# EPICS alarm handler configuration: mps_database/bare/alarms/areas/mpln_sps_mp03.alhConfig
GROUP NULL MPLN:SPS:MP03:1
$ALIAS MPS Link Node 193
$GUIDANCE
LTUH MPS
   Group Name: MPLN:SPS:MP03:1
   Summary PV:  MPLN:SPS:MP03:1:STATSUMY
$END
CHANNEL  MPLN:SPS:MP03:1    MPLN:SPS:MP03:1:MPS_EN_RBV		-----
CHANNEL  MPLN:SPS:MP03:1    MPLN:SPS:MP03:1:LC1_MODE_RBV		-----
